Staubli VAL3: start.pgx

program start()
begin
  taskCreateSync "motion", 0.05, bMotionOverrun, motionControl()
end
